INTERFACE ITF_BaseLogger_Item

METHOD PUBLIC GetID : UINT
VAR_INPUT
END_VAR
END_METHOD

METHOD GetInformationToDisplayEvent : ST_BaseLogger_ItemDataToDisplay
VAR_INPUT
	uiIDEvent				: UINT;
END_VAR
END_METHOD

END_INTERFACE

(* stored: Version 1.1.0.1
   Itf ITF_BaseLogger_Item: Id {9acb94a3-79f9-0d22-1a7a-50b9e1991d9a}
   Method GetID: Id {94ee4911-8643-0cde-2f4d-b033ebc42178}
   Method GetInformationToDisplayEvent: Id {93fc010a-fb9f-082f-1e1f-a9126d7f1608} *)
